Staubli VAL3: AdvanceSingal.pgx

program AdvanceSingal()
begin
  //需要提前开启的信号

end
